Universal Robots PolyScope program: fillWater.urp

Program fillWater (installation=20240827 directory=/programs/Demos/water createdIn=5.15.1 lastSavedIn=5.15.1 robotSerialNumber=20245500285)
Calibrated DH parameters: a=[0.000097, -0.210459, -0.026602, 0.000137, 0.000078, 0]; d=[0.162601, 254.180657, -54.076236, -199.970743, 0.099615, 0.099684]; alpha=[1.569796, -0.001455, 0.001957, 1.570525, -1.571561, 0]; deltaTheta=[0, -1.053331, 8.839472, -1.50296, 0.000002, 0]
InitVariablesNode
Robot Program (runOnlyOnce=false)
  Script: usb = rpc_factory("xmlrpc","http://192.168.1.7:9120/RPC2")
  MoveJ speed 60 deg/s, acceleration 80 deg/s^2 (useActiveTCP=true) feature=Base
    Waypoint 路点_1: TCP in base x=431.817 y=-466.748 z=371.687 mm, rx=-0.0114 ry=1.57 rz=0.0102 rad; joints [90.581, -84.024, 117.141, -123.16, 0.001, 0] deg; TCP offset x=-0.17 y=0 z=192.95 mm, rx=0 ry=0 rz=0 rad
  counter := 0
  'show'
  If False
    Popup Message (haltProgram=false message=12 inputType=Text)
    Script: usb.open()
    Popup Message (haltProgram=false message=12 inputType=Text)
    Script: usb.adaptiveClose()
  'fill'
  Popup Message (haltProgram=false message=12 inputType=Text)
  Script: usb.open()
  Popup Message (haltProgram=false message=12 inputType=Text)
  Script: usb.adaptiveClose()
  SuppressedNode
    Script: usb.adaptiveFillWater()
  Script: usb.fillwater()
  SuppressedNode
    Loop Forever
      SuppressedNode
        Wait Sleep waitTime=0.01
      Script: counter=counter+1
  Popup Message (haltProgram=false message=12 inputType=Text)
  Script: usb.open()
